Universal Robots URScript: 20240920_mediapipe.script

def P20240920_mediapipe():
  global _hidden_verificationVariable=0
  set_target_payload(1.500000, [0.001000, -0.003000, 0.050000], [0.003026, 0.003026, 0.003026, 0.000000, 0.000000, 0.000000])
  set_tcp(p[-1.7E-4,0.0,0.19294999999999998,0.0,0.0,0.0])
  set_tool_communication(True, 115200, 0, 1, 1.5, 3.5)
  set_tool_output_mode(0)
  set_tool_digital_output_mode(0, 1)
  set_tool_digital_output_mode(1, 1)
  set_tool_voltage(24)
  set_standard_analog_input_domain(0, 1)
  set_standard_analog_input_domain(1, 1)
  set_tool_analog_input_domain(0, 1)
  set_tool_analog_input_domain(1, 1)
  set_analog_outputdomain(0, 1)
  set_analog_outputdomain(1, 0)
  set_input_actions_to_default()
  set_tool_digital_input_action(0, "freedrive")
  set_gravity([0.0, 0.0, 9.82])
  set_safety_mode_transition_hardness(0)
  global i_var_1=p[0.31, 0, 0, 0, 0, 0]
  global u24179u38754_1=p[0.0,0.0,0.0,0.0,0.0,0.0]
  global u24179u38754_2=p[0.2,0.6,0.4,-1.4839444017850547,-0.07419722008925289,-2.225916602677581]
  global u24179u38754_3=p[0.1459477485431481,-0.10308445883660293,0.13857682671027435,-0.008977024873201634,0.014216906208388691,-2.4400986907073663]
  global u28857_1=p[0.10203918836050063,-0.5259531579406657,0.376430278847906,-0.18768520041296463,-3.1325095402283982,-0.09669790600413578]
  global u28857_2=p[0.0665007526844362,-0.3872123180436422,0.638459113340625,-0.320095108678139,-2.6903368475934015,1.4700117755369673]
  global u30452u32447_1=p[0.0,0.0,0.0,0.0,0.0,0.0]
  step_count_b4d2483f_8893_49b8_936f_64b158deedd3 = 0.0
  thread Step_Counter_Thread_a2b80ebc_5de6_4f94_bd03_a8c00072d35d():
    while (True):
      step_count_b4d2483f_8893_49b8_936f_64b158deedd3 = step_count_b4d2483f_8893_49b8_936f_64b158deedd3 + 1.0
      sync()
    end
  end
  run Step_Counter_Thread_a2b80ebc_5de6_4f94_bd03_a8c00072d35d()
  global u36335u28857_1_p=p[.083397192482, -.466994623149, .106166314196, -2.221436009358, -2.221414367123, .000061766622]
  global u36335u28857_1_q=[1.4604315757751465, -1.5431790848127385, 2.045967404042379, -2.074360509912008, -1.5714219252215784, 1.463240623474121]
  $ 2 "开始前"
  $ 3 "MoveJ"
  $ 4 "路点_1" "breakAfter"
  movej(u36335u28857_1_q, a=0.6981317007977318, v=0.8726646259971648)
  $ 5 "joints≔get_actual_joint_positions()"
  global joints=get_actual_joint_positions()
  $ 7 "home≔get_actual_tcp_pose()"
  global home= get_actual_tcp_pose ()
  $ 8 "write_output_boolean_register(0, False )"
  write_output_boolean_register(0,  False  )
  $ 10 "等待: 0.01"
  sleep(0.01)
  $ 11 "popup('Registers reset, run PC code and then click Continue',title='Hi Daniel',blocking= True )"
  popup("Registers reset, run PC code and then click Continue",title="Hi Daniel",blocking=  True  )
  $ 12 "mode≔0"
  global mode=0
  $ 27 "Thread_1"
  thread Thread_1():
    while (True):
      $ 28 "tmp≔p[0,0,0,0,0,0]"
      global tmp=p[0,0,0,0,0,0]
      $ 29 "循环"
      while (True):
        $ 30 "脚本: pose_register.script"
        tmp[0]=read_input_float_register(0)
        tmp[1]=read_input_float_register(1)
        tmp[2]=read_input_float_register(2)
        tmp[3]=read_input_float_register(3)
        tmp[4]=read_input_float_register(4)
        tmp[5]=read_input_float_register(5)
        $ 31 "joints≔get_inverse_kin(p[tmp[0],tmp[1],tmp[2],tmp[3],tmp[4],tmp[5]],get_actual_joint_positions())"
        global joints= get_inverse_kin (p[tmp[0],tmp[1],tmp[2],tmp[3],tmp[4],tmp[5]],get_actual_joint_positions())
        $ 32 "sync()"
        sync()
        $ 33 "mode≔read_input_integer_register(0)"
        global mode=read_input_integer_register(0)
        $ 34 "sync()"
        sync()
      end
    end
  end
  threadId_Thread_1 = run Thread_1()
  while (True):
    $ 13 "机器人程序"
    $ 14 "write_output_boolean_register(0, True )"
    write_output_boolean_register(0,  True  )
    $ 15 "sync()"
    sync()
    $ 16 "循环 mode<3"
    while (mode<3):
      $ 17 "循环 mode≟1"
      while (mode == 1):
        $ 18 "MoveJ"
        $ 19 "joints" "breakAfter"
        movej(joints, a=1.3962634015954636, v=1.0471975511965976)
        $ 20 "write_output_boolean_register(0, False )"
        write_output_boolean_register(0,  False  )
        $ 21 "sync()"
        sync()
      end
      $ 22 "循环 mode≟2"
      while (mode == 2):
        $ 23 "servoj(joints, 0, 0, 0.03, 0.9, 1800)"
        servoj(joints, 0, 0, 0.03, 0.9, 1800)
      end
      $ 24 "循环 mode≟3"
      while (mode == 3):
        $ 25 "中止"
        halt
      end
    end
    $ 26 "sync()"
    sync()
  end
end
